// TIA Portal V19 export
DATA_BLOCK "iDB_TimeCounterPause"   // DB71
{ DB_Accessible_From_OPC_UA := 'FALSE' }
// stored: AutoNumber false, DBAccessibleFromOPCUA false, DBAccessibleFromWebserver false, InstanceOfName FB_TimeCounter, InstanceOfType FB
"FB_TimeCounter"
   // VAR_INPUT
   //    xClockSecond { ExternalAccessible := 'False'; ExternalVisible := 'False'; ExternalWritable := 'False'} : Bool;
   //    xStart { ExternalAccessible := 'False'; ExternalVisible := 'False'; ExternalWritable := 'False'} : Bool;
   //    xStop { ExternalAccessible := 'False'; ExternalVisible := 'False'; ExternalWritable := 'False'} : Bool;
   //    xResetCounter { ExternalAccessible := 'False'; ExternalVisible := 'False'; ExternalWritable := 'False'} : Bool;
   // END_VAR
   // VAR_OUTPUT
   //    PerpetualCounter { ExternalAccessible := 'False'; ExternalVisible := 'False'; ExternalWritable := 'False'} : UDInt;
   //    "Counter" { ExternalAccessible := 'False'; ExternalVisible := 'False'; ExternalWritable := 'False'} : UDInt;
   // END_VAR
   // VAR
   //    sxEnableCount { ExternalAccessible := 'False'; ExternalVisible := 'False'; ExternalWritable := 'False'} : Bool;
   //    sxFpStart { ExternalAccessible := 'False'; ExternalVisible := 'False'; ExternalWritable := 'False'} : Bool;
   //    sxFpStop { ExternalAccessible := 'False'; ExternalVisible := 'False'; ExternalWritable := 'False'} : Bool;
   // END_VAR
   // VAR RETAIN
   //    miDB_Counter { ExternalAccessible := 'False'; ExternalVisible := 'False'; ExternalWritable := 'False'; S7_SetPoint := 'True'} : CTU_UDINT;
   //    miDB_PerpetualCount { ExternalAccessible := 'False'; ExternalVisible := 'False'; ExternalWritable := 'False'; S7_SetPoint := 'True'} : CTU_UDINT;
   // END_VAR
   // VAR
   //    sxFpResetCounter { ExternalAccessible := 'False'; ExternalVisible := 'False'; ExternalWritable := 'False'} : Bool;
   //    sxResetCounter { ExternalAccessible := 'False'; ExternalVisible := 'False'; ExternalWritable := 'False'} : Bool;
   // END_VAR
BEGIN
END_DATA_BLOCK
